(*
SPDX-FileCopyrightText: © 2026 Oleksandr Tiutyk <trofimich@gmail.com>
SPDX-License-Identifier: MIT
License: https://opensource.org/license/mit
*)

(*!
<summary>
Beckhoff EL2409: 16-channel HD digital output terminal (24 V DC, 0.5 A, protected).
</summary>
<description>
Process image mapping structure for the high-density EL2409 EtherCAT terminal with 16 discrete 24 V DC 0.5 A
outputs with electronic protection.
When used for I/O, link located fields or their containing buffers to the matching selected PDOs.
The record is not a packed wire buffer; compiler padding is not part of the device specification.
Unlinked/default values do not prove valid I/O. The caller evaluates bus/channel validity before use.
Use one owner task per instance and externally synchronize other access; multi-field snapshots are not atomic.
Copies store data without creating hardware links. Keep borrowed field references valid while consumers are bound.
This passive record performs no validation, synchronization, configuration or protocol advancement.
</description>
*)
TYPE EL2409 :
STRUCT
	Ch01 AT %Q* : BOOL;
	Ch02 AT %Q* : BOOL;
	Ch03 AT %Q* : BOOL;
	Ch04 AT %Q* : BOOL;
	Ch05 AT %Q* : BOOL;
	Ch06 AT %Q* : BOOL;
	Ch07 AT %Q* : BOOL;
	Ch08 AT %Q* : BOOL;
	Ch09 AT %Q* : BOOL;
	Ch10 AT %Q* : BOOL;
	Ch11 AT %Q* : BOOL;
	Ch12 AT %Q* : BOOL;
	Ch13 AT %Q* : BOOL;
	Ch14 AT %Q* : BOOL;
	Ch15 AT %Q* : BOOL;
	Ch16 AT %Q* : BOOL;
END_STRUCT
END_TYPE

(* stored: Version 1.1.0.1, ProductVersion 3.1.4026.20
   DUT EL2409: Id {e22845a2-a54f-4241-bad9-8a91a7c30578} *)
